{attribute addProperty BoxType "EL5101-0000-0001"}
{attribute addProperty Id "InputsAT %I*Inputs_6F37F4E44050OutputsAT %Q*Outputs_4D4E89362430WcStateAT %I*WcState_F855686C1620InfoDataAT %I*InfoData_BC63D37F80100"}
{attribute addProperty CRC "693920209"}
{attribute addProperty SizeInBites "160"}
{attribute addProperty SizeInBytes "20"}
TYPE EL5101_D480A6FC :
STRUCT
	{attribute addProperty Name "Inputs"}
	Inputs : Inputs_6F37F4E4;
	{attribute addProperty Name "Outputs"}
	Outputs : Outputs_4D4E8936;
	{attribute addProperty Name "WcState"}
	WcState : WcState_F855686C;
	{attribute addProperty Name "InfoData"}
	InfoData : InfoData_BC63D37F;
END_STRUCT
END_TYPE

(* stored: Version 1.2.0.0, ProductVersion 3.1.4024.9
   DUT EL5101_D480A6FC: Id {e4919717-ec01-410f-9aa4-c674fb5e8c8e} *)
